Staubli VAL3: start.pgx

program start()
begin

  nTest[0] = 0
  nTest[1] = 2
  nTest[2] = -4
  nTest[3] = 10
  nTest[5] = -3
  nTest[6] = 4

  call rollsum(nTest, 3,nResultTest)

end
